// TIA Portal V20 export
TYPE "typeCmControlNode"
// stored: Namespace Unit1.Em8
   STRUCT
      interlock : "Unit1.Em8.typeCmControlNodeInterlock";
      command : "Unit1.Em8.typeCmControlNodeCommand";
      softcam : "Unit1.Em8.typeCmControlNodeSoftCam";
      brakeTest : "Unit1.Em8.typeCmControlNodeBrakeTest";
   END_STRUCT;
END_TYPE
